// Mitsubishi GX Works2 project: plc16 read   PLC: FX3G

// global labels: Global1
VAR_GLOBAL
  Start_switch AT X007 : BOOL;
  System_on AT Y007 : BOOL;
  Lack_material AT M0 : BOOL;
  Emergency_switch AT X005 : BOOL;
  Analog_output AT D8282 : INT;
  Total_boxes AT D1100 : REAL;
  Raspberry_input AT D1120 : REAL;
  Lemon_inpout AT D1130 : REAL;
  Stabilizer_input AT D1140 : REAL;
  Bears_input AT D1150 : REAL;
  Raspberry_amount AT D1160 : REAL;
  Lemon_amount AT D1170 : REAL;
  Stabilizer_amount AT D1180 : REAL;
  Bears_amount AT D1190 : REAL;
  Make_iceCream AT X001 : BOOL;
  Analog_input1 AT D8280 : INT;
  Analog_value AT D2000 : REAL;
END_VAR
VAR_GLOBAL CONSTANT
  divide_num : REAL := 400;
  Pinuk_LB : REAL := 6;
  Regular_UB : REAL := 5;
END_VAR
VAR_GLOBAL
  Pinuk_selected AT M1 : BOOL;
  Regular_selected AT M2 : BOOL;
END_VAR
VAR_GLOBAL CONSTANT
  Raspberry_regular_LB : REAL := 280;
  Lemon_regular_LB : REAL := 455;
  Bears_regular_LB : REAL := 28;
END_VAR
VAR_GLOBAL
  Regular_check AT M3 : BOOL;
  Flag_RR AT M10 : BOOL;
  Flag_BR AT M12 : BOOL;
  Flag_LR AT M11 : BOOL;
END_VAR
VAR_GLOBAL CONSTANT
  Stabilizer_regular_LB : REAL := 105;
END_VAR
VAR_GLOBAL
  Flag_SR AT M13 : BOOL;
END_VAR
VAR_GLOBAL CONSTANT
  Raspberry_Pinuk_LB : REAL := 385;
END_VAR
VAR_GLOBAL
  Flag_RP AT M20 : BOOL;
END_VAR
VAR_GLOBAL CONSTANT
  Lemon_Pinuk_LB : REAL := 665;
END_VAR
VAR_GLOBAL
  Flag_LP AT M21 : BOOL;
END_VAR
VAR_GLOBAL CONSTANT
  Bears_Pinuk_LB : REAL := 70;
END_VAR
VAR_GLOBAL
  Flag_BP AT M22 : BOOL;
END_VAR
VAR_GLOBAL CONSTANT
  Stabilizer_Pinuk_LB : REAL := 210;
END_VAR
VAR_GLOBAL
  Flag_SP AT M23 : BOOL;
  Pinuk_check AT M4 : BOOL;
  Raspberry_iceCream AT D2100 : REAL;
END_VAR
VAR_GLOBAL CONSTANT
  Regular_RQ : REAL := 350;
END_VAR
VAR_GLOBAL
  Lemon_iceCream AT D2110 : REAL;
END_VAR
VAR_GLOBAL CONSTANT
  Regular_LQ : REAL := 490;
  Pinuk_RQ : REAL := 560;
  Pinuk_LQ : REAL := 700;
END_VAR
VAR_GLOBAL
  Make_Light AT TS1 : BOOL;
  TC_1 AT TC1 : BOOL;
END_VAR
VAR_GLOBAL CONSTANT
  Timer_light_iceCream : INT := 50;
END_VAR
VAR_GLOBAL
  IceCream_light AT Y000 : BOOL;
  Finish1_flag AT M24 : BOOL;
  Cool_iceCream AT X002 : BOOL;
  Raspberry_cool AT D2120 : REAL;
  Lemon_cool AT D2130 : REAL;
  Temp_sensor AT X003 : BOOL;
  Cool_light AT Y002 : BOOL;
  Cool_timer AT TS2 : BOOL;
  TC_2 AT TC2 : BOOL;
END_VAR
VAR_GLOBAL CONSTANT
  Timer_light_cool : INT := 80;
END_VAR
VAR_GLOBAL
  Cool_flag AT TS2 : BOOL;
  Finish2_flag AT M25 : BOOL;
  Mix_iceCream AT D2200 : REAL;
  Flicker AT M30 : BOOL;
  TC_3 AT TC3 : BOOL;
END_VAR
VAR_GLOBAL CONSTANT
  Regular_mixTime : INT := 30;
END_VAR
VAR_GLOBAL
  TS_3 AT TS3 : BOOL;
  Y_5 AT Y005 : BOOL;
END_VAR
VAR_GLOBAL CONSTANT
  Flick_time : INT := 5;
END_VAR
VAR_GLOBAL
  TC_4 AT TC4 : BOOL;
  TS_4 AT TS4 : BOOL;
  Y_6 AT Y006 : BOOL;
END_VAR
VAR_GLOBAL CONSTANT
  ResetCon : BOOL;
  Flick_time_regular : INT := 30;
  Flick_time_pinuk : INT := 50;
  blink_time : INT := 5;
END_VAR
VAR_GLOBAL
  blink_flag AT M31 : BOOL;
  TC_5 AT TC5 : BOOL;
  TC_6 AT TC6 : BOOL;
  TS_5 AT TS5 : BOOL;
  TS_6 AT TS6 : BOOL;
END_VAR
VAR_GLOBAL CONSTANT
  Rest_con : BOOL;
END_VAR
VAR_GLOBAL
  Finish3_flag AT M31 : BOOL;
  Start_packing AT X004 : BOOL;
  con_packing AT X000 : BOOL;
  packing_light AT Y004 : BOOL;
  one_con_start AT CC1 : BOOL;
END_VAR
VAR_GLOBAL CONSTANT
  one_con_packed : INT := 1;
END_VAR
VAR_GLOBAL
  Seven_con_end AT CC2 : BOOL;
END_VAR
VAR_GLOBAL CONSTANT
  seven_con_packed : INT := 7;
END_VAR
VAR_GLOBAL
  first_con AT CS1 : BOOL;
  seven_con AT CS2 : BOOL;
  packing_process AT Y004 : BOOL;
  end_packing AT M40 : BOOL;
END_VAR
VAR_GLOBAL CONSTANT
  add_package : REAL := 1;
  mul_num : REAL := 40;
END_VAR

// task Task_01 (event TRUE, interval 0, priority 31): POU_01

PROGRAM POU_01
(* structured ladder/FBD written out as ST: instructions are called as NAME(EN, inputs, outputs); _pN, _eN, _tN stand for wires *)
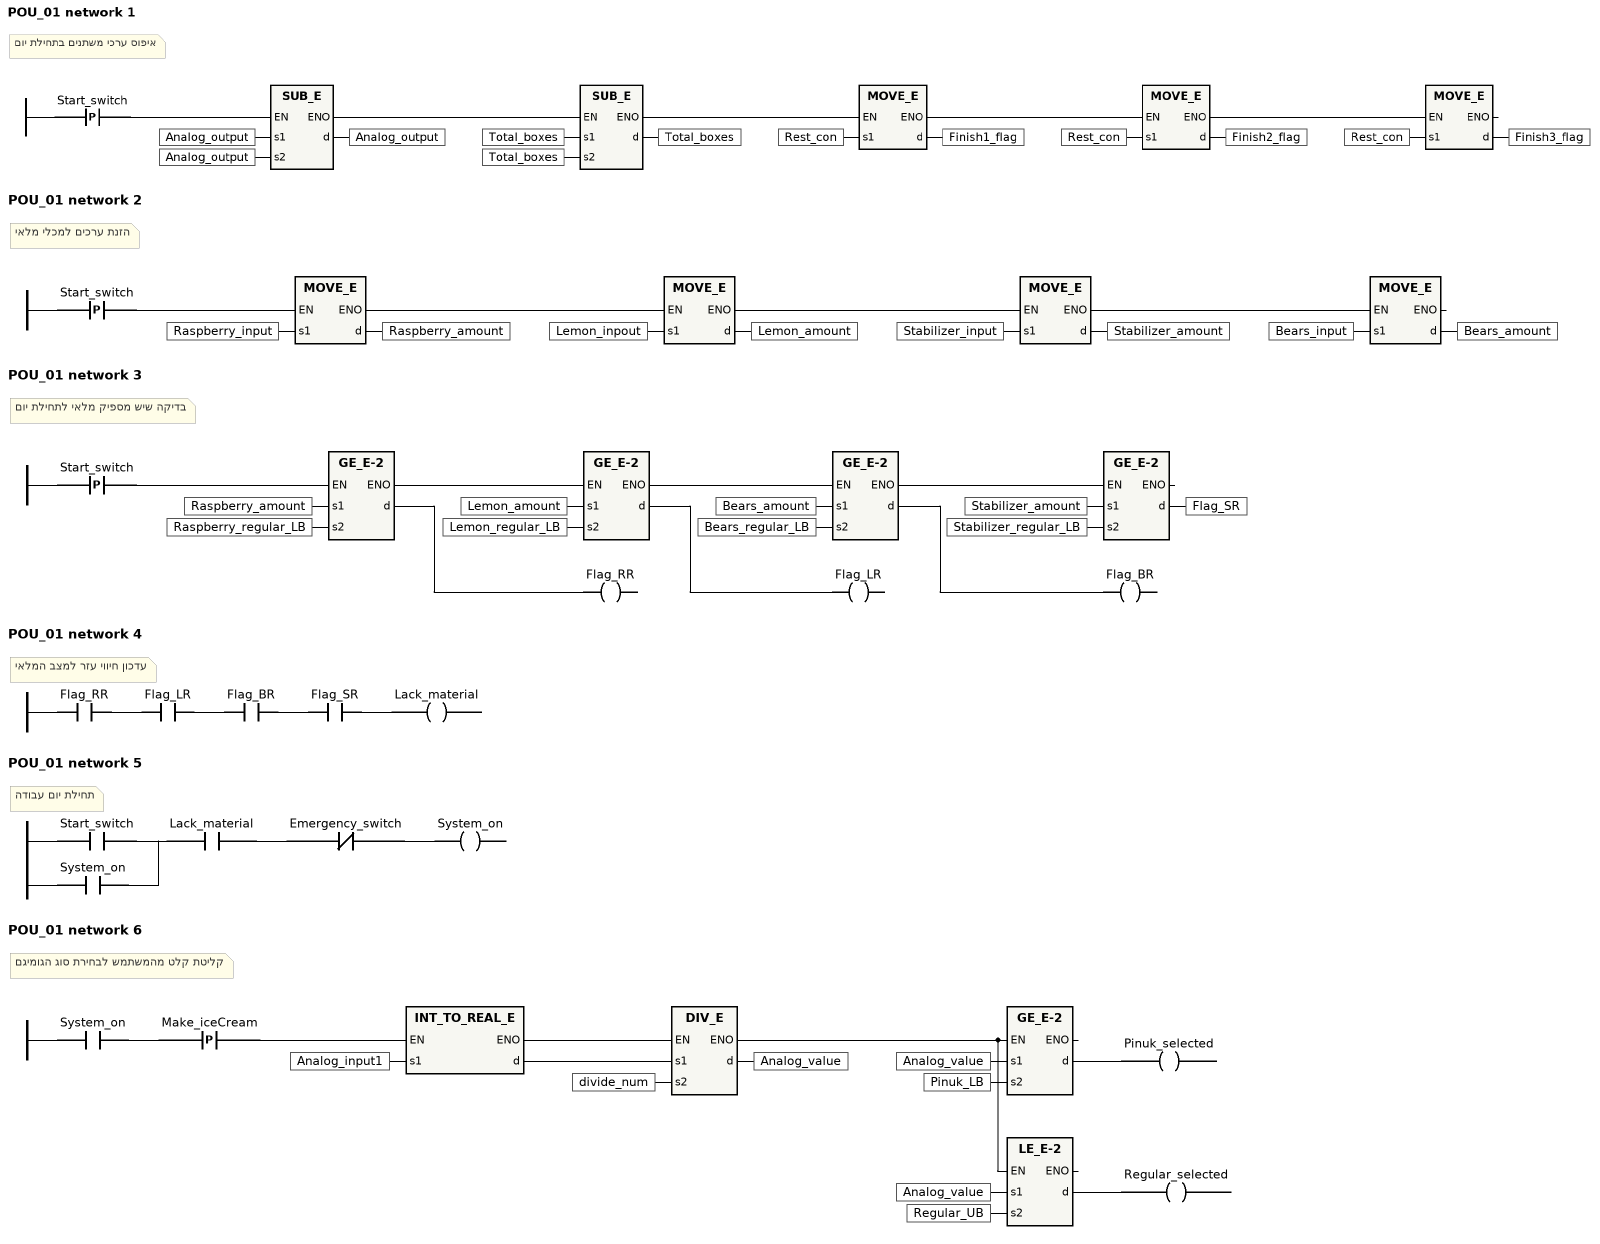
(* network 1 *)
(* איפוס ערכי משתנים בתחילת יום *)
_e1 := SUB_E(LDP(TRUE, Start_switch), Analog_output, Analog_output, Analog_output);
_e2 := SUB_E(_e1, Total_boxes, Total_boxes, Total_boxes);
_e3 := MOVE_E(_e2, Rest_con, Finish1_flag);
_e4 := MOVE_E(_e3, Rest_con, Finish2_flag);
MOVE_E(_e4, Rest_con, Finish3_flag);
(* network 2 *)
(* הזנת ערכים למכלי מלאי *)
_e1 := MOVE_E(LDP(TRUE, Start_switch), Raspberry_input, Raspberry_amount);
_e2 := MOVE_E(_e1, Lemon_inpout, Lemon_amount);
_e3 := MOVE_E(_e2, Stabilizer_input, Stabilizer_amount);
MOVE_E(_e3, Bears_input, Bears_amount);
(* network 3 *)
(* בדיקה שיש מספיק מלאי לתחילת יום *)
_e2 := GE_E(LDP(TRUE, Start_switch), Raspberry_amount, Raspberry_regular_LB, _t1);
_e4 := GE_E(_e2, Lemon_amount, Lemon_regular_LB, _t3);
_e6 := GE_E(_e4, Bears_amount, Bears_regular_LB, _t5);
GE_E(_e6, Stabilizer_amount, Stabilizer_regular_LB, Flag_SR);
Flag_RR := _t1;
Flag_LR := _t3;
Flag_BR := _t5;
(* network 4 *)
(* עדכון חיווי עזר למצב המלאי *)
Lack_material := Flag_RR AND Flag_LR AND Flag_BR AND Flag_SR;
(* network 5 *)
(* תחילת יום עבודה *)
System_on := ((Start_switch OR System_on) AND Lack_material) AND NOT Emergency_switch;
(* network 6 *)
(* קליטת קלט מהמשתמש לבחירת סוג הגומיגם *)
_e2 := INT_TO_REAL_E(System_on AND LDP(TRUE, Make_iceCream), Analog_input1, _t1);
_e3 := DIV_E(_e2, _t1, divide_num, Analog_value);
GE_E(_e3, Analog_value, Pinuk_LB, _t4);
Pinuk_selected := _t4;
LE_E(_e3, Analog_value, Regular_UB, _t5);
Regular_selected := _t5;
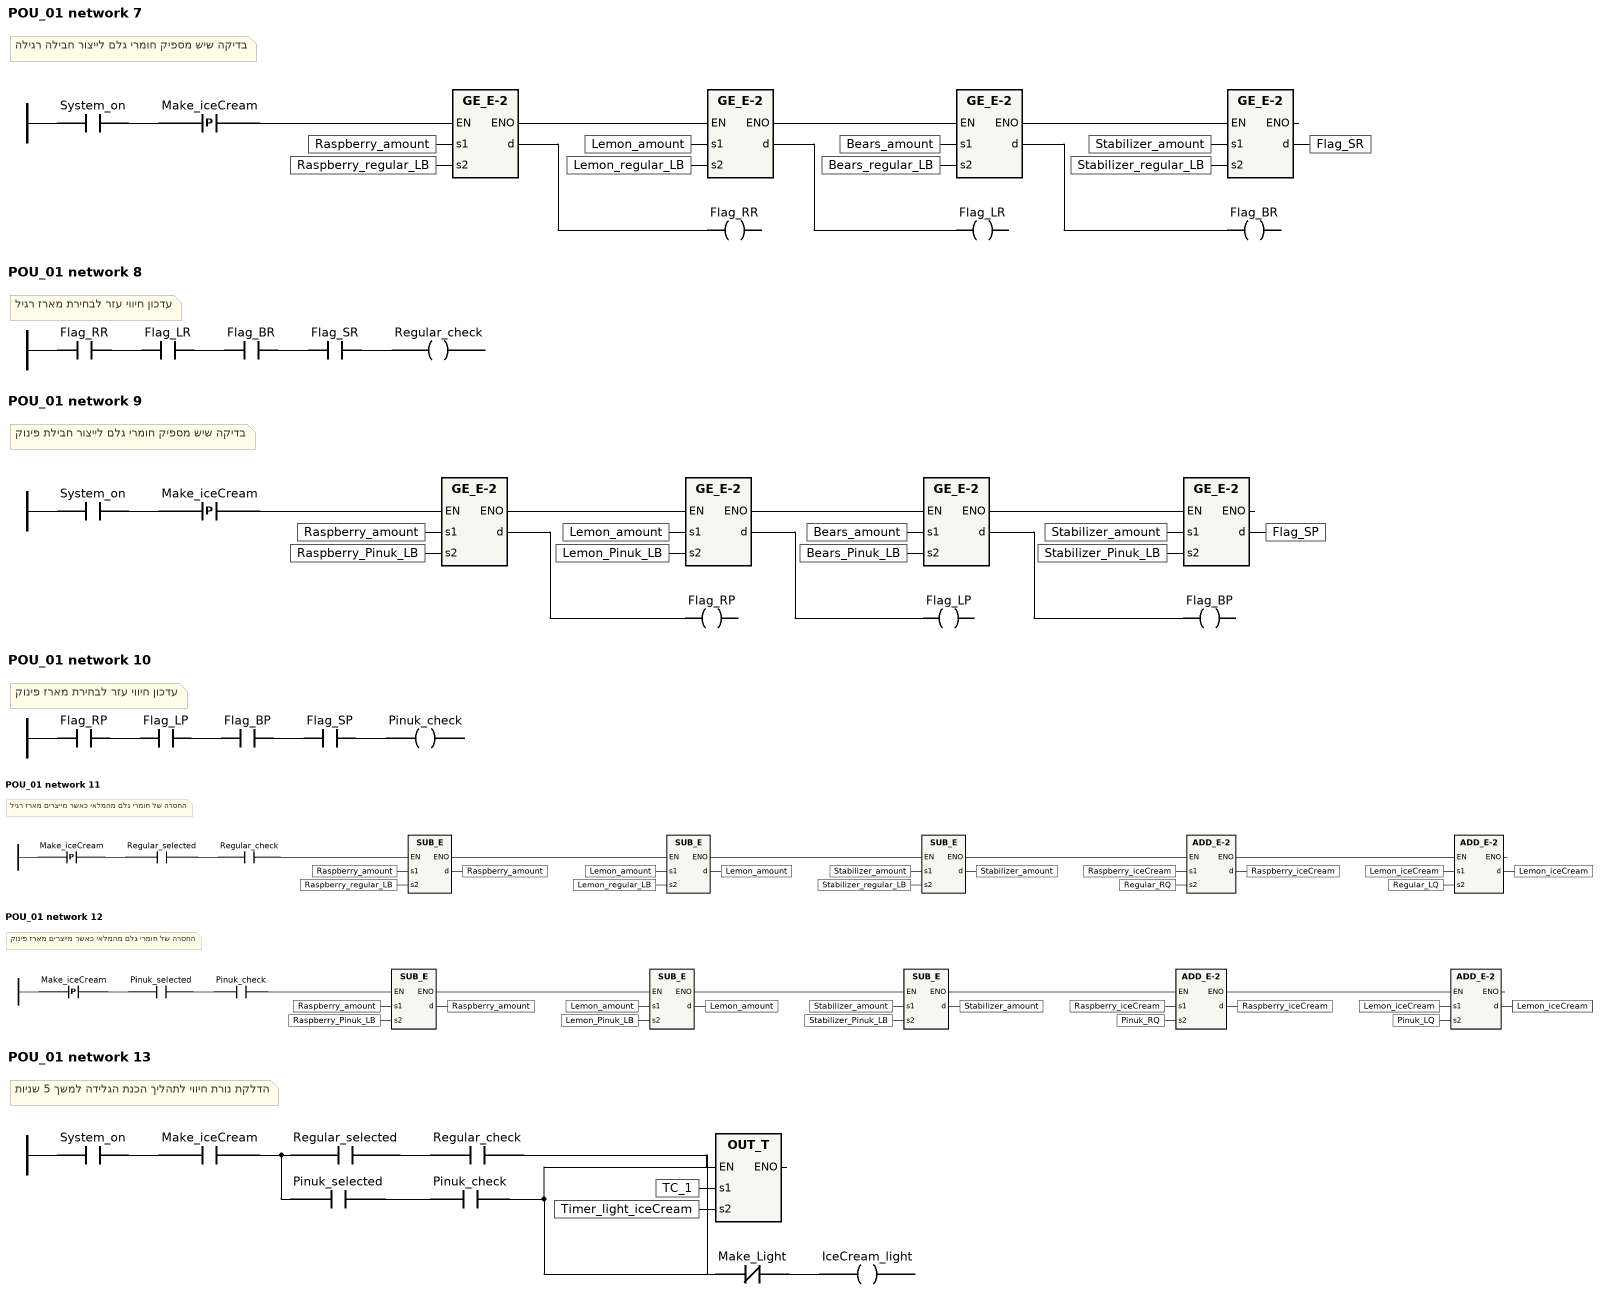
(* network 7 *)
(* בדיקה שיש מספיק חומרי גלם לייצור חבילה רגילה *)
_e2 := GE_E(System_on AND LDP(TRUE, Make_iceCream), Raspberry_amount, Raspberry_regular_LB, _t1);
_e4 := GE_E(_e2, Lemon_amount, Lemon_regular_LB, _t3);
_e6 := GE_E(_e4, Bears_amount, Bears_regular_LB, _t5);
GE_E(_e6, Stabilizer_amount, Stabilizer_regular_LB, Flag_SR);
Flag_RR := _t1;
Flag_LR := _t3;
Flag_BR := _t5;
(* network 8 *)
(* עדכון חיווי עזר לבחירת מארז רגיל *)
Regular_check := Flag_RR AND Flag_LR AND Flag_BR AND Flag_SR;
(* network 9 *)
(* בדיקה שיש מספיק חומרי גלם לייצור חבילת פינוק *)
_e2 := GE_E(System_on AND LDP(TRUE, Make_iceCream), Raspberry_amount, Raspberry_Pinuk_LB, _t1);
_e4 := GE_E(_e2, Lemon_amount, Lemon_Pinuk_LB, _t3);
_e6 := GE_E(_e4, Bears_amount, Bears_Pinuk_LB, _t5);
GE_E(_e6, Stabilizer_amount, Stabilizer_Pinuk_LB, Flag_SP);
Flag_RP := _t1;
Flag_LP := _t3;
Flag_BP := _t5;
(* network 10 *)
(* עדכון חיווי עזר לבחירת מארז פינוק *)
Pinuk_check := Flag_RP AND Flag_LP AND Flag_BP AND Flag_SP;
(* network 11 *)
(* החסרה של חומרי גלם מהמלאי כאשר מייצרים מארז רגיל *)
_e1 := SUB_E(LDP(TRUE, Make_iceCream) AND Regular_selected AND Regular_check, Raspberry_amount, Raspberry_regular_LB, Raspberry_amount);
_e2 := SUB_E(_e1, Lemon_amount, Lemon_regular_LB, Lemon_amount);
_e3 := SUB_E(_e2, Stabilizer_amount, Stabilizer_regular_LB, Stabilizer_amount);
_e4 := ADD_E(_e3, Raspberry_iceCream, Regular_RQ, Raspberry_iceCream);
ADD_E(_e4, Lemon_iceCream, Regular_LQ, Lemon_iceCream);
(* network 12 *)
(* החסרה של חומרי גלם מהמלאי כאשר מייצרים מארז פינוק *)
_e1 := SUB_E(LDP(TRUE, Make_iceCream) AND Pinuk_selected AND Pinuk_check, Raspberry_amount, Raspberry_Pinuk_LB, Raspberry_amount);
_e2 := SUB_E(_e1, Lemon_amount, Lemon_Pinuk_LB, Lemon_amount);
_e3 := SUB_E(_e2, Stabilizer_amount, Stabilizer_Pinuk_LB, Stabilizer_amount);
_e4 := ADD_E(_e3, Raspberry_iceCream, Pinuk_RQ, Raspberry_iceCream);
ADD_E(_e4, Lemon_iceCream, Pinuk_LQ, Lemon_iceCream);
(* network 13 *)
(* הדלקת נורת חיווי לתהליך הכנת הגלידה למשך 5 שניות *)
_p1 := System_on AND Make_iceCream;
_p2 := (_p1 AND Regular_selected AND Regular_check) OR (_p1 AND Pinuk_selected AND Pinuk_check);
IceCream_light := _p2 AND NOT Make_Light;
OUT_T(_p2, TC_1, Timer_light_iceCream);
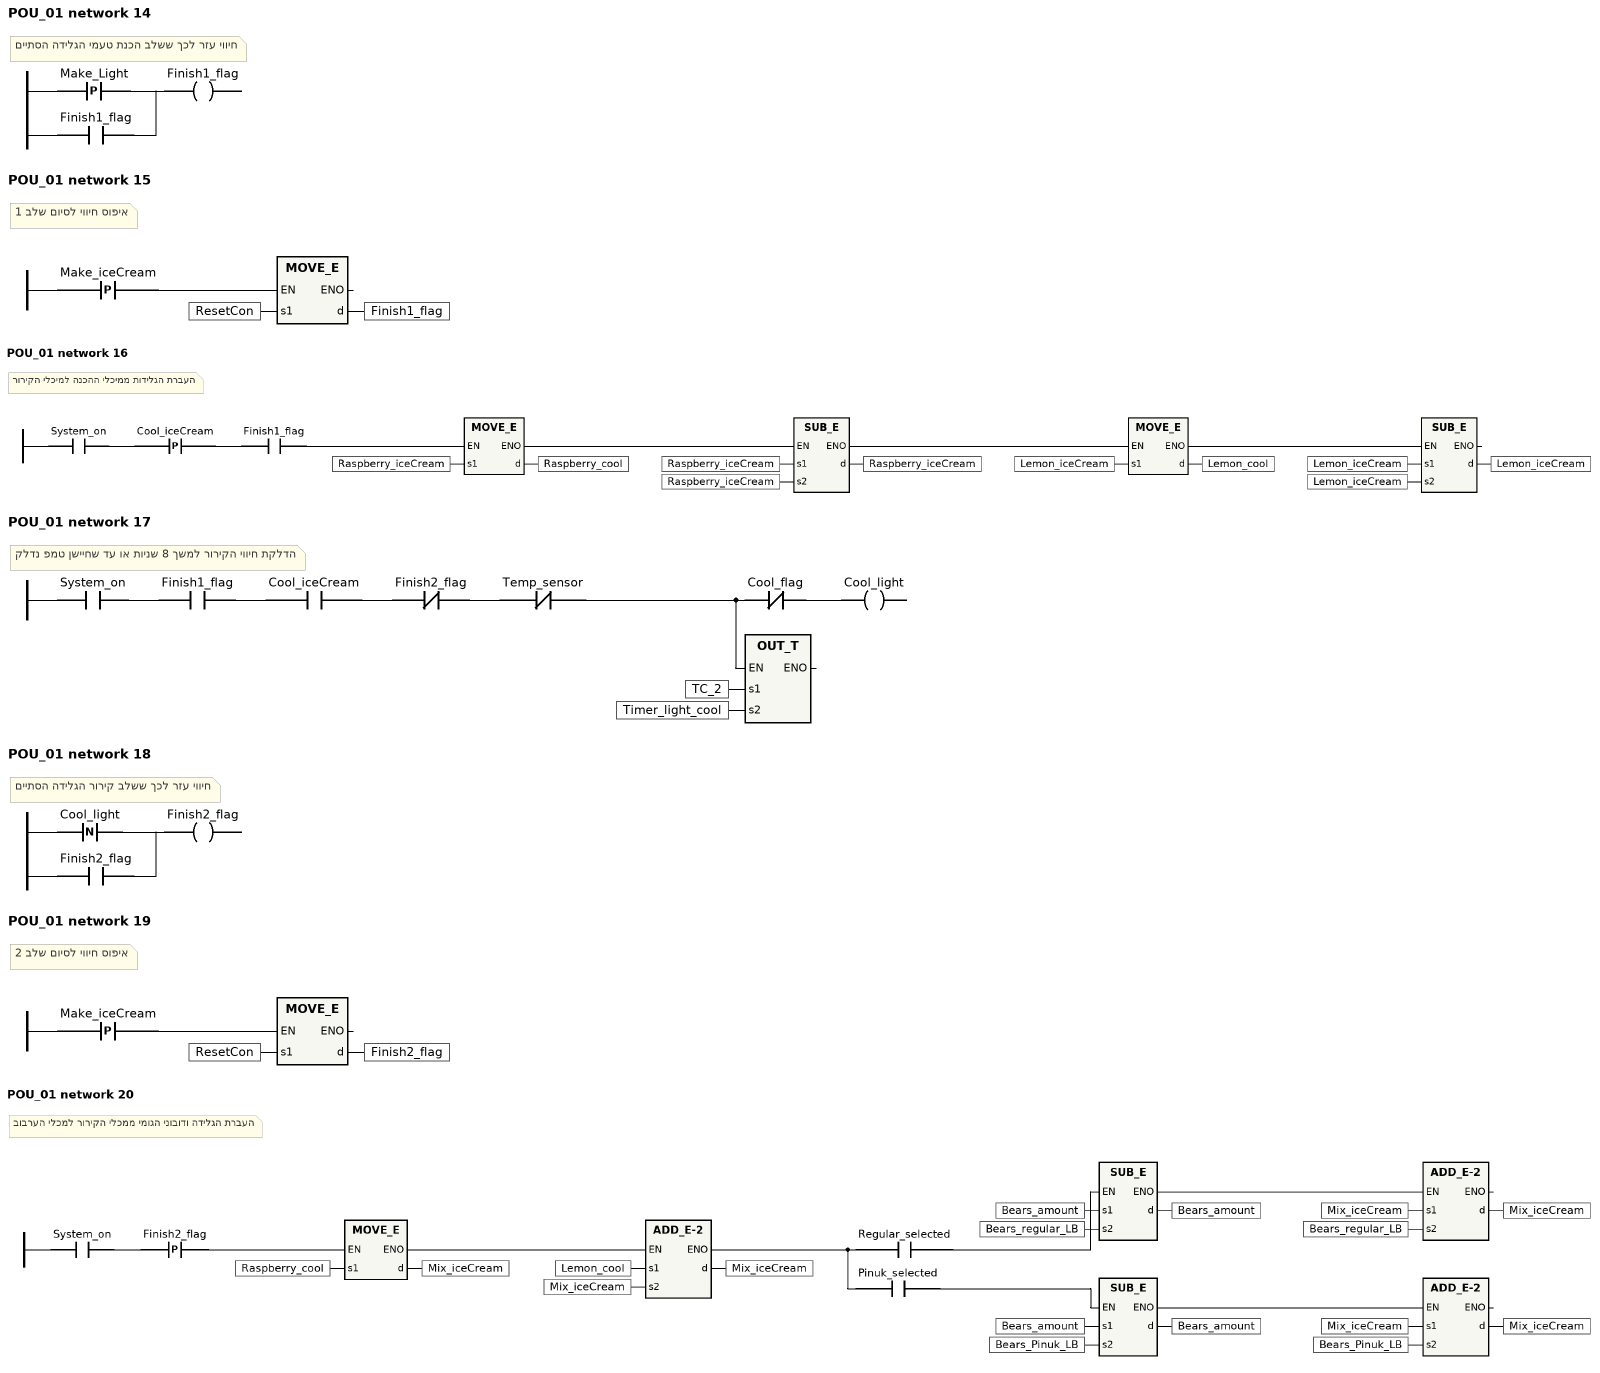
(* network 14 *)
(* חיווי עזר לכך ששלב הכנת טעמי הגלידה הסתיים *)
Finish1_flag := LDP(TRUE, Make_Light) OR Finish1_flag;
(* network 15 *)
(* איפוס חיווי לסיום שלב 1 *)
MOVE_E(LDP(TRUE, Make_iceCream), ResetCon, Finish1_flag);
(* network 16 *)
(* העברת הגלידות ממיכלי ההכנה למיכלי הקירור *)
_e1 := MOVE_E(System_on AND LDP(TRUE, Cool_iceCream) AND Finish1_flag, Raspberry_iceCream, Raspberry_cool);
_e2 := SUB_E(_e1, Raspberry_iceCream, Raspberry_iceCream, Raspberry_iceCream);
_e3 := MOVE_E(_e2, Lemon_iceCream, Lemon_cool);
SUB_E(_e3, Lemon_iceCream, Lemon_iceCream, Lemon_iceCream);
(* network 17 *)
(* הדלקת חיווי הקירור למשך 8 שניות או עד שחיישן טמפ נדלק *)
_p1 := System_on AND Finish1_flag AND Cool_iceCream AND NOT Finish2_flag AND NOT Temp_sensor;
Cool_light := _p1 AND NOT Cool_flag;
OUT_T(_p1, TC_2, Timer_light_cool);
(* network 18 *)
(* חיווי עזר לכך ששלב קירור הגלידה הסתיים *)
Finish2_flag := LDF(TRUE, Cool_light) OR Finish2_flag;
(* network 19 *)
(* איפוס חיווי לסיום שלב 2 *)
MOVE_E(LDP(TRUE, Make_iceCream), ResetCon, Finish2_flag);
(* network 20 *)
(* העברת הגלידה ודובוני הגומי ממכלי הקירור למכלי הערבוב *)
_e1 := MOVE_E(System_on AND LDP(TRUE, Finish2_flag), Raspberry_cool, Mix_iceCream);
_e2 := ADD_E(_e1, Lemon_cool, Mix_iceCream, Mix_iceCream);
_e3 := SUB_E(_e2 AND Regular_selected, Bears_amount, Bears_regular_LB, Bears_amount);
ADD_E(_e3, Mix_iceCream, Bears_regular_LB, Mix_iceCream);
_e4 := SUB_E(_e2 AND Pinuk_selected, Bears_amount, Bears_Pinuk_LB, Bears_amount);
ADD_E(_e4, Mix_iceCream, Bears_Pinuk_LB, Mix_iceCream);
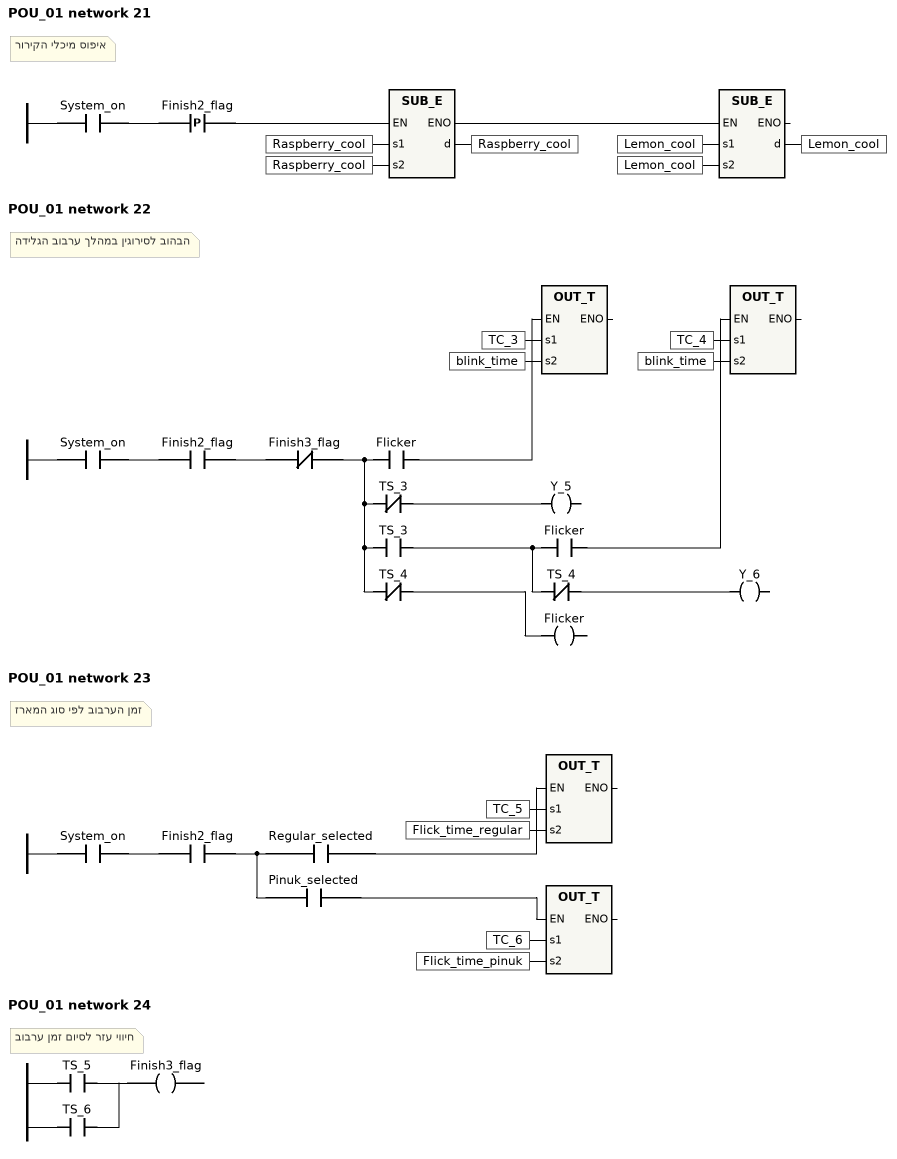
(* network 21 *)
(* איפוס מיכלי הקירור *)
_e1 := SUB_E(System_on AND LDP(TRUE, Finish2_flag), Raspberry_cool, Raspberry_cool, Raspberry_cool);
SUB_E(_e1, Lemon_cool, Lemon_cool, Lemon_cool);
(* network 22 *)
(* הבהוב לסירוגין במהלך ערבוב הגלידה *)
_p1 := System_on AND Finish2_flag AND NOT Finish3_flag;
OUT_T(_p1 AND Flicker, TC_3, blink_time);
Y_5 := _p1 AND NOT TS_3;
_p2 := _p1 AND TS_3;
OUT_T(_p2 AND Flicker, TC_4, blink_time);
Y_6 := _p2 AND NOT TS_4;
Flicker := _p1 AND NOT TS_4;
(* network 23 *)
(* זמן הערבוב לפי סוג המארז *)
_p1 := System_on AND Finish2_flag;
OUT_T(_p1 AND Regular_selected, TC_5, Flick_time_regular);
OUT_T(_p1 AND Pinuk_selected, TC_6, Flick_time_pinuk);
(* network 24 *)
(* חיווי עזר לסיום זמן ערבוב *)
Finish3_flag := TS_5 OR TS_6;
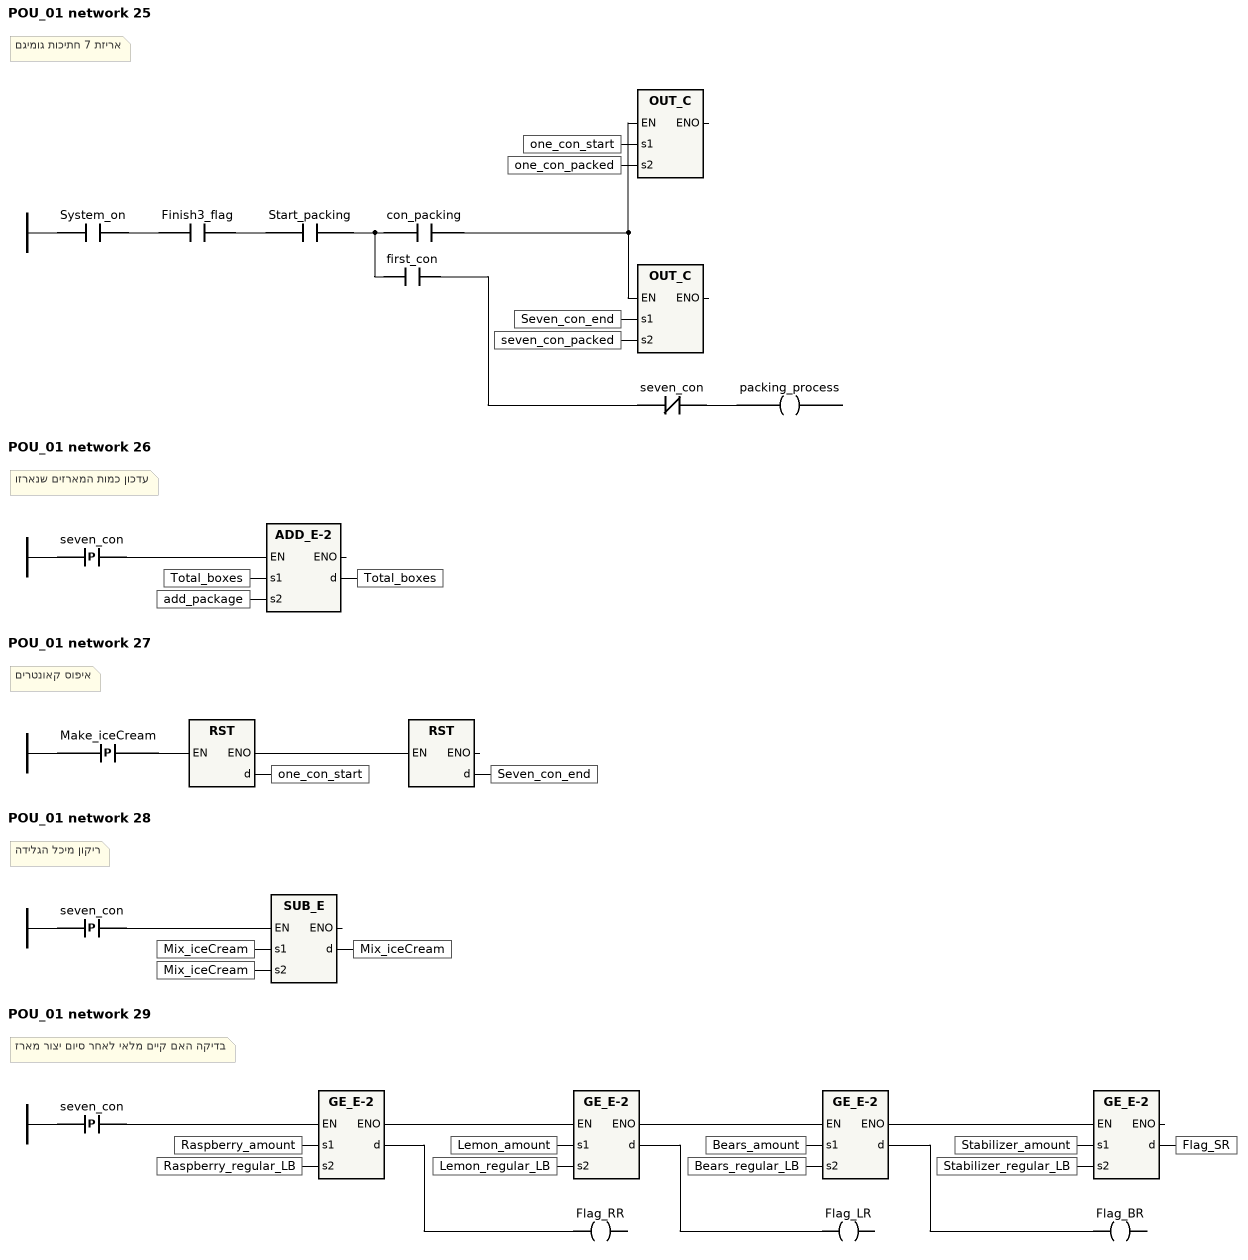
(* network 25 *)
(* אריזת 7 חתיכות גומיגם *)
_p1 := System_on AND Finish3_flag AND Start_packing;
_p2 := _p1 AND con_packing;
OUT_C(_p2, one_con_start, one_con_packed);
OUT_C(_p2, Seven_con_end, seven_con_packed);
packing_process := _p1 AND first_con AND NOT seven_con;
(* network 26 *)
(* עדכון כמות המארזים שנארזו *)
ADD_E(LDP(TRUE, seven_con), Total_boxes, add_package, Total_boxes);
(* network 27 *)
(* איפוס קאונטרים *)
_e1 := RST(LDP(TRUE, Make_iceCream), one_con_start);
RST(_e1, Seven_con_end);
(* network 28 *)
(* ריקון מיכל הגלידה *)
SUB_E(LDP(TRUE, seven_con), Mix_iceCream, Mix_iceCream, Mix_iceCream);
(* network 29 *)
(* בדיקה האם קיים מלאי לאחר סיום יצור מארז *)
_e2 := GE_E(LDP(TRUE, seven_con), Raspberry_amount, Raspberry_regular_LB, _t1);
_e4 := GE_E(_e2, Lemon_amount, Lemon_regular_LB, _t3);
_e6 := GE_E(_e4, Bears_amount, Bears_regular_LB, _t5);
GE_E(_e6, Stabilizer_amount, Stabilizer_regular_LB, Flag_SR);
Flag_RR := _t1;
Flag_LR := _t3;
Flag_BR := _t5;
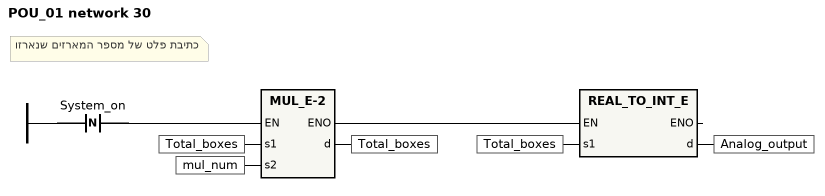
(* network 30 *)
(* כתיבת פלט של מספר המארזים שנארזו *)
_e1 := MUL_E(LDF(TRUE, System_on), Total_boxes, mul_num, Total_boxes);
REAL_TO_INT_E(_e1, Total_boxes, Analog_output);
END_PROGRAM
